PROGRAM ArmMove
VAR
	
	point												:Points;					// 当前腕关节坐标
	target_angle										:Angles;					// 臂左右电机目标角度
	manualState											:USINT;						// 手动控制状态标志位，0
	speed												:REAL := 1;					// 笛卡尔坐标位移速度
	x													:REAL;						// 腕关节目标位置x
	y													:REAL;						// 腕关节目标位置y
	wrist_angle											:REAL;
	wrist_MoveAbs										:MC_MoveAbsolute;
	
	LeftArm_Right_ExtPosGen_Enable						:MC_ExtSetPointGenEnable;
	LeftArm_Right_ExtPosGen_Disable                     :MC_ExtSetPointGenDisable;
	LeftArm_Left_ExtPosGen_Enable                       :MC_ExtSetPointGenEnable;
	LeftArm_Left_ExtPosGen_Disable	                    :MC_ExtSetPointGenDisable;
	
	fb_SerialCom		:FB_SerialCom;					//串口
	wrist_angle_int		:INT;
	wrist_angle_byte	:BYTE;
	
	
END_VAR

axis_LeftArm_Left();
axis_LeftArm_Right();
ExtPosGen();

// 外部位置发生器失能
LeftArm_Right_ExtPosGen_Enable.Execute 		:= FALSE;
LeftArm_Right_ExtPosGen_Disable.Execute 	:= FALSE;
LeftArm_Left_ExtPosGen_Enable.Execute 		:= FALSE;
LeftArm_Left_ExtPosGen_Disable.Execute 		:= FALSE;

IF bManualCtrl_Asm_LeftArm THEN
	
	// 运动学正解出当前腕关节点坐标
	point := ArmFK(axis_LeftArm_Right.NcToPlc.ActPos, axis_LeftArm_Left.NcToPlc.ActPos);
	
	// 用舵机进行程序验证的串口背景通讯
	//BackgroundSerialCtrl();
	
	IF bAutoCtrl_Part_LeftWrist THEN
		
		wrist_angle := WristIK(point.x, point.y);		// 逆解出腕电机角度
		wrist_angle_int:= TO_INT(wrist_angle);
		
		// 用舵机进行程序验证的串口测试
		//wrist_angle_byte:= INT_TO_BYTE(wrist_angle_int);
		//fb_SerialCom(TxBuffer:= TxBuffer, RxBuffer:= RxBuffer, angle:= wrist_angle_byte);	
		
		wrist_MoveAbs(Axis:= axis_LeftArm_Wrist, Execute:= TRUE, Position:= wrist_angle, Velocity:= 5, Acceleration:= 10, Deceleration:= , Jerk:= , BufferMode:= , 
					  Options:= , Done=> , Busy=> , Active=> , CommandAborted=> , Error=> , ErrorID=> );		// 腕电机走绝对定位
	END_IF
	

	IF bLeftArm_Forward THEN
		x := point.x;
		y := point.y + speed;
		target_angle := ArmIK(x, y);
		manualState := 1;
		
	ELSIF bLeftArm_Backward THEN
	
		x := point.x;
		y := point.y - speed;
		target_angle := ArmIK(x, y);
		manualState := 1;
		
	ELSIF bLeftArm_Left THEN
		
		x := point.x - speed;
		y := point.y;
		target_angle := ArmIK(x, y);
		manualState := 1;
		
	ELSIF bLeftArm_Right THEN
		
		x := point.x + speed;
		y := point.y;
		target_angle := ArmIK(x, y);
		manualState := 1;
		
	ELSE
		manualState := 0;
	END_IF
	
	
	
	CASE manualState OF
		0:
			LeftArm_Right_ExtPosGen_Enable.Execute 		:= FALSE;
			LeftArm_Right_ExtPosGen_Disable.Execute 	:= TRUE;
			LeftArm_Left_ExtPosGen_Enable.Execute 		:= FALSE;
			LeftArm_Left_ExtPosGen_Disable.Execute 		:= TRUE;
		
		1:
			LeftArm_Right_ExtPosGen_Enable.Execute := TRUE;
			LeftArm_Left_ExtPosGen_Enable.Execute := TRUE;
			IF axis_LeftArm_Right.Status.ExtSetPointGenEnabled AND axis_LeftArm_Left.Status.ExtSetPointGenEnabled THEN
				MC_ExtSetPointGenFeed(
					Position:= target_angle.theta1_right, 
					Velocity:= 30,  
					Acceleration:= 10,  
					Direction:= 1, 
					Axis:= axis_LeftArm_Right);
		
				MC_ExtSetPointGenFeed(
					Position:= target_angle.theta2_left, 
					Velocity:= 30,  
					Acceleration:= 10,  
					Direction:= 1, 
					Axis:= axis_LeftArm_Left);
			END_IF
	END_CASE

//ELSE

END_IF

ACTION ExtPosGen:
LeftArm_Right_ExtPosGen_Enable(
	Axis:= axis_LeftArm_Right, 
	Execute:= LeftArm_Right_ExtPosGen_Enable.Execute, 
	Position:= , 
	PositionType:= , 
	Done=> , 
	Busy=> , 
	Error=> , 
	ErrorID=> , 
	Enabled=> );
	
LeftArm_Right_ExtPosGen_Disable(
	Axis:= axis_LeftArm_Right, 
	Execute:= LeftArm_Right_ExtPosGen_Disable.Execute, 
	Done=> , 
	Busy=> , 
	Error=> , 
	ErrorID=> , 
	Enabled=> );
	
LeftArm_Left_ExtPosGen_Enable(
	Axis:= axis_LeftArm_Left, 
	Execute:= LeftArm_Left_ExtPosGen_Enable.Execute, 
	Position:= , 
	PositionType:= , 
	Done=> , 
	Busy=> , 
	Error=> , 
	ErrorID=> , 
	Enabled=> );
	
LeftArm_Left_ExtPosGen_Disable(
	Axis:= axis_LeftArm_Left, 
	Execute:= LeftArm_Left_ExtPosGen_Disable.Execute, 
	Done=> , 
	Busy=> , 
	Error=> , 
	ErrorID=> , 
	Enabled=> );
END_ACTION

END_PROGRAM

(* stored: Version 1.1.0.1, ProductVersion 3.1.4024.14
   POU ArmMove: Id {82e9130f-3eaf-4158-9f64-c53d364c6ee4}, SpecialFunc None
   Action ExtPosGen: Id {b057b60f-3c1a-48f8-86ef-b3bf94d37dff} *)
